{attribute addProperty BoxType "KL9999"}
{attribute addProperty Id "Channel_1Channel_22349BF100"}
{attribute addProperty CRC "3125334992"}
{attribute addProperty SizeInBites "0"}
{attribute addProperty SizeInBytes "0"}
TYPE KL9999_BA48D3D0 :
STRUCT
	{attribute addProperty Name "Channel_1"}
	Channel_1 : Channel_22349BF1;
END_STRUCT
END_TYPE

(* stored: Version 1.2.0.0, ProductVersion 3.1.4024.9
   DUT KL9999_BA48D3D0: Id {09e3a2de-2db1-4293-9e46-423de8d694f3} *)
